FUNCTION FC_Check_SOH : BOOL
VAR_INPUT
	I_sString : REFERENCE TO T_MaxString;
END_VAR
VAR
	stringPos	: INT;
END_VAR

stringPos := FIND(I_sString, SOH);
IF stringPos <> 0 THEN
	I_sString := MID(I_sString, LEN(I_sString), stringPos+1);
	FC_Check_SOH := TRUE;
ELSE
	FC_Check_SOH := FALSE;
END_IF

END_FUNCTION

(* stored: Version 1.1.0.1, ProductVersion 3.1.4024.15
   POU FC_Check_SOH: Id {2d688172-31e2-4996-9bc1-3f6b7c237b20}, SpecialFunc None *)
